//---------------------------------------------------------------------------------------------------------------
//
//  HAUD 2024.04.16
//
//
//
//---------------------------------------------------------------------------------------------------------------
// This SOFTWARE is provided as an Exemple by THE PROVIDER "as is" and "with all faults." THE PROVIDER makes no 
// representations or warranties of any kind concerning the safety, suitability, lack of viruses, inaccuracies, 
// typographical errors, or other harmful components of this SOFTWARE. There are inherent dangers in the use of 
// any software, and you are solely responsible for determining whether this SOFTWARE is compatible with your 
// equipment and other software installed on your equipment. You are also solely responsible for the protection 
// of your equipment and backup of your data, and THE PROVIDER will not be liable for any damages you may suffer 
// in connection with using, modifying, or distributing this SOFTWARE.
//---------------------------------------------------------------------------------------------------------------
FUNCTION_BLOCK fb_Mover
VAR
  _nMoverId         : UINT;

  _sState           : STRING;

  _Mover            : REFERENCE TO Tc3_Mc3PlanarMotion.MC_PlanarMover;
  _Feedback         : REFERENCE TO Tc3_Mc3PlanarMotion.MC_PlanarFeedback;

  // mover compact axis information
  _stInfo           : REFERENCE TO ST_MOVER_INFO; // ActPos, Enable, ...

  _bError           : BOOL;   // used in Cycle()
  _nErrorIdMover,             // used in Cycle()
  _nErrorIdPower    : UDINT;  // used in Cycle()

  //---------------------------------------------------------------------------
  // 
  //---------------------------------------------------------------------------
  _wMoverState      : DWORD;

END_VAR

METHOD Check : BOOL
// check The thing that should not be

IF NOT (_nMoverId > 0)
THEN
  _sState                     := 'Mover: missing ID';
  RETURN;
END_IF

IF NOT __ISVALIDREF(_Mover)
THEN
  _sState                     := 'Mover: missing pointer';
  RETURN;
END_IF

IF NOT __ISVALIDREF(_stInfo)
THEN
  _sState                     := '_stInfo: missing pointer';
  RETURN;
END_IF

_sState                       := 'CHECK_DONE';
Check                         := TRUE;
END_METHOD

METHOD Cycle : E_PROGRESS
VAR_INST
  _eState             : E_PROGRESS;

  _rtrigMoverError,
  _rtrigPowerError    : Tc2_Standard.R_TRIG;
END_VAR
IF NOT Check() THEN Cycle := E_PROGRESS.PROGRESS_ERROR; RETURN; END_IF

//-----------------------------------------------------------------------------------------------
// cyclic NC mapping
//-----------------------------------------------------------------------------------------------
_Mover.Update();
_Feedback.Update();
//-----------------------------------------------------------------------------------------------


//-----------------------------------------------------------------------------------------------
// cyclic error
//-----------------------------------------------------------------------------------------------

_rtrigPowerError(CLK := _Feedback.Error);

IF _rtrigMoverError.Q
THEN
  _bError                 := TRUE;  // deleted by Reset()
  // catch error
  _nErrorIdMover          := _Feedback.ErrorId;
  _stInfo.nErrorId        := _nErrorIdMover;
END_IF
//-----------------------------------------------------------------------------------------------

//-----------------------------------------------------------------------------------------------
// cyclic state
//-----------------------------------------------------------------------------------------------
IF NOT (_Mover.MCTOPLC.STD.State = MC_PLANAR_STATE.Enabled)
THEN
  _eState                       := E_PROGRESS.PROGRESS_INIT;
ELSE
  _eState                       := E_PROGRESS.PROGRESS_WORKING;
END_IF
 
IF _bError
THEN
  _eState                       := E_PROGRESS.PROGRESS_ERROR;
END_IF
//-----------------------------------------------------------------------------------------------


//-----------------------------------------------------------------------------
// cyclic Mover info data
// get collision avoiding information from cyclic interface
//-----------------------------------------------------------------------------------------------
_stInfo.bMoverEnabled           := (_Mover.MCTOPLC.STD.State = MC_PLANAR_STATE.Enabled);
_stInfo.bMoverStandstill        := NOT (_Mover.MCTOPLC.STD.Busy.BusyXYC);
_stInfo.bMoverError             := _bError;

_stInfo.rActPos.x               := _Mover.MCTOPLC.ACT.ActPos.x;
_stInfo.rActPos.y               := _Mover.MCTOPLC.ACT.ActPos.y;
_stInfo.rActPos.c               := _Mover.MCTOPLC.ACT.ActPos.c;
                                
_stInfo.rActPosX                := _Mover.MCTOPLC.ACT.ActPos.x;
_stInfo.rActPosY                := _Mover.MCTOPLC.ACT.ActPos.y;
_stInfo.rActPosC                := _Mover.MCTOPLC.ACT.ActPos.c;
                                
_stInfo.rActPosZ                := _Mover.MCTOPLC.ACT.ActPos.z;
                                
_stInfo.rActVeloX               := _Mover.MCTOPLC.ACT.ActVelo.x;
_stInfo.rActVeloY               := _Mover.MCTOPLC.ACT.ActVelo.y;
_stInfo.rActVeloZ               := _Mover.MCTOPLC.ACT.ActVelo.z;
_stInfo.rActVeloC               := _Mover.MCTOPLC.ACT.ActVelo.c;
//-----------------------------------------------------------------------------

Cycle                           := _eState;
END_METHOD

METHOD Disable : E_PROGRESS
VAR_INPUT
  Execute             : BOOL;
END_VAR
VAR_INST
  _nErrorId           : UDINT;
  _eState             : E_PROGRESS;
END_VAR
IF NOT Execute THEN _eState  := E_PROGRESS.PROGRESS_INIT; END_IF 
IF NOT Check() THEN Disable  := E_PROGRESS.PROGRESS_ERROR; RETURN; END_IF


CASE _eState
OF
  E_PROGRESS.PROGRESS_INIT:
    IF Execute
    THEN
      _nErrorId               := 0;
      _eState                 := E_PROGRESS.PROGRESS_BUSY;
    END_IF
END_CASE
//-----------------------------------------------------------------------------
//-----------------------------------------------------------------------------
CASE _eState
OF
  E_PROGRESS.PROGRESS_BUSY:
    _eState                   := E_PROGRESS.PROGRESS_PREPARE;
    _Mover.Disable(_Feedback);
END_CASE
//-----------------------------------------------------------------------------
//-----------------------------------------------------------------------------
CASE _eState
OF
  E_PROGRESS.PROGRESS_PREPARE:
    IF (_Mover.MCTOPLC.STD.State = MC_PLANAR_STATE.Disabled)
    THEN
      IF _Feedback.Error
      THEN
        _eState                 := E_PROGRESS.PROGRESS_ERROR;
      ELSIF _Feedback.Done
      THEN
        _eState                 := E_PROGRESS.PROGRESS_DONE;
      END_IF
    END_IF
END_CASE
//-----------------------------------------------------------------------------
//-----------------------------------------------------------------------------

Disable                       := _eState;
END_METHOD

METHOD Enable : E_PROGRESS
VAR_INPUT
  Execute             : BOOL;
END_VAR
VAR_INST
  _nErrorId           : UDINT;
  _eState             : E_PROGRESS;
END_VAR
IF NOT Execute THEN _eState  := E_PROGRESS.PROGRESS_INIT; END_IF 
IF NOT Check() THEN Enable   := E_PROGRESS.PROGRESS_ERROR; RETURN; END_IF


CASE _eState
OF
  E_PROGRESS.PROGRESS_INIT:
    IF Execute
    THEN
      _nErrorId               := 0;
      _eState                 := E_PROGRESS.PROGRESS_BUSY;
    END_IF
END_CASE
//-----------------------------------------------------------------------------
//-----------------------------------------------------------------------------
CASE _eState
OF
  E_PROGRESS.PROGRESS_BUSY:
    _eState                   := E_PROGRESS.PROGRESS_PREPARE;
    _Mover.Enable(_Feedback);
END_CASE
//-----------------------------------------------------------------------------
//-----------------------------------------------------------------------------
CASE _eState
OF
  E_PROGRESS.PROGRESS_PREPARE:
    IF (_Mover.MCTOPLC.STD.State = MC_PLANAR_STATE.Enabled)
    THEN
      IF _Feedback.Error
      THEN
        _eState                 := E_PROGRESS.PROGRESS_ERROR;
      ELSIF _Feedback.Done
      THEN
        _eState                 := E_PROGRESS.PROGRESS_DONE;
      END_IF
    ELSIF (_Mover.MCTOPLC.STD.State = MC_PLANAR_STATE.Error)
    THEN
      _eState                   := E_PROGRESS.PROGRESS_ERROR;
    END_IF
END_CASE
//-----------------------------------------------------------------------------
//-----------------------------------------------------------------------------

Enable                   := _eState;
END_METHOD

PROPERTY Feedback : reference to Tc3_Mc3PlanarMotion.MC_PlanarFeedback
SET
_Feedback REF= Feedback;
END_SET
END_PROPERTY

METHOD Halt : E_PROGRESS
VAR_INPUT
  Execute             : BOOL;
  stMoveData          : ST_MOVE_DATA;
END_VAR
VAR_INST
  _nErrorId           : UDINT;
  _eState             : E_PROGRESS;

	_Position           : Tc3_Physics.PositionXYC;
	_Constraint         : Tc3_Physics.DynamicConstraint_PathXY;
	_Options            : Tc3_Mc3PlanarMotion.ST_MoveToPositionOptions;
	_OptionsC           : ST_MoveCOptions;
END_VAR
IF NOT Execute 
THEN 
	_eState := E_PROGRESS.PROGRESS_INIT; 
END_IF 
IF NOT Check() 
THEN 
	Halt := E_PROGRESS.PROGRESS_ERROR; 
	RETURN; 
END_IF


CASE _eState
OF
  E_PROGRESS.PROGRESS_INIT:
    IF Execute
    THEN
      _nErrorId               := 0;
      _eState                 := E_PROGRESS.PROGRESS_BUSY;
    END_IF
END_CASE
//-----------------------------------------------------------------------------
//-----------------------------------------------------------------------------
CASE _eState
OF
  E_PROGRESS.PROGRESS_BUSY:
    _eState                     := E_PROGRESS.PROGRESS_PREPARE;
		_Position.SetValuesXYC(
                            x   := stMoveData.rPos.x,
													  y   := stMoveData.rPos.y,
                            c	  := 0.0);
								
		_Constraint.SetValuesVADJ(
                            V   := stMoveData.rVelo, 
                            A   := stMoveData.rAcc, 
                            D   := stMoveData.rAcc, 
                            J   := stMoveData.rJerk);

		_Options.useOrientation	    := FALSE;
END_CASE
//-----------------------------------------------------------------------------
//-----------------------------------------------------------------------------
CASE _eState
OF
  E_PROGRESS.PROGRESS_PREPARE:
    _eState                     := E_PROGRESS.PROGRESS_STARTUP;
    _Mover.Halt(_Feedback, _Constraint); 
END_CASE
//-----------------------------------------------------------------------------
//-----------------------------------------------------------------------------
CASE _eState
OF
  E_PROGRESS.PROGRESS_STARTUP:
    IF _Feedback.Error
    THEN
      _nErrorId                 := _feedback.ErrorId;
      _stInfo.nErrorId          := _nErrorId;

      _eState                   := E_PROGRESS.PROGRESS_ERROR;
    ELSIF _Feedback.Done
    THEN
      _eState                   := E_PROGRESS.PROGRESS_DONE;
    END_IF
END_CASE
//-----------------------------------------------------------------------------
//-----------------------------------------------------------------------------

Halt                          := _eState;
END_METHOD

PROPERTY Mover : REFERENCE to Tc3_Mc3PlanarMotion.MC_PlanarMover
SET
_Mover REF= Mover;
END_SET
END_PROPERTY

PROPERTY MoverId : uint
SET
_nMoverId := MoverId;
END_SET
END_PROPERTY

PROPERTY MoverInfo : REFERENCE to ST_MOVER_INFO
SET


	_stInfo ref= MoverInfo;
END_SET
END_PROPERTY

METHOD MoveToPos : E_PROGRESS
VAR_INPUT
  Execute             : BOOL;
  stMoveData          : ST_MOVE_DATA;
END_VAR
VAR_INST
  _nErrorId           : UDINT;
  _rDelta,
  _rPos               : LREAL;
  _eState             : E_PROGRESS;

	_Position           : Tc3_Physics.PositionXYC;
	_Constraint         : Tc3_Physics.DynamicConstraint_PathXY;
  _ConstraintC        : Tc3_Physics.DynamicConstraint_PathXY;
	_Options            : Tc3_Mc3PlanarMotion.ST_MoveToPositionOptions;
	_OptionsC           : ST_MoveCOptions;

  _rTmpV,
  _rTmpA,
  _rTmpD,
  _rTmpJ              : LREAL;
END_VAR
IF NOT Execute THEN _eState  := E_PROGRESS.PROGRESS_INIT; END_IF 
IF NOT Check() THEN MoveToPos   := E_PROGRESS.PROGRESS_ERROR; RETURN; END_IF


CASE _eState
OF
  E_PROGRESS.PROGRESS_INIT:
    IF Execute
    THEN
      _nErrorId                 := 0;
      _rDelta                   := SEL((stMoveData.rDelta < 0.01), stMoveData.rDelta, 0.05);
      _eState                   := E_PROGRESS.PROGRESS_BUSY;

      _rTmpV   := stMoveData.rVelo/10.0; 
      _rTmpA   := stMoveData.rAcc/10.0;
      _rTmpD   := stMoveData.rAcc/10.0; 
      _rTmpJ   := stMoveData.rJerk/10.0;


		  _Constraint.SetValuesVADJ(
                            V   := _rTmpV, 
                            A   := _rTmpA, 
                            D   := _rTmpD, 
                            J   := _rTmpJ);
  
      _Mover.MoveZ(
            commandFeedback     := _Feedback, 
            targetPosition      := stMoveData.rPosZ,
            constraint          := _Constraint);

		  _Options.useOrientation	  := FALSE;
    END_IF
END_CASE
//-----------------------------------------------------------------------------
//-----------------------------------------------------------------------------
CASE _eState
OF
  E_PROGRESS.PROGRESS_BUSY:
    IF _Feedback.Error OR _Feedback.Aborted
    THEN
      _nErrorId                 := _feedback.ErrorId;
      _stInfo.nErrorId          := _nErrorId;

      _eState                   := E_PROGRESS.PROGRESS_ERROR;

    ELSIF _Feedback.Done OR NOT _Feedback.Busy
    THEN
      _eState                   := E_PROGRESS.PROGRESS_PREPARE;

      IF (stMoveData.nAxisFirst = 1)
      THEN
        _Position.SetValuesXYC(
                            x   := stMoveData.rPos.x,
                            y   := _Mover.MCTOPLC.SET.SetPos.y,
                            c	  := 0.0);

      ELSIF (stMoveData.nAxisFirst = 2)
      THEN
        _Position.SetValuesXYC(
                            x   := _Mover.MCTOPLC.SET.SetPos.x,
                            y   := stMoveData.rPos.y,
                            c	  := 0.0);
      ELSE
        _Position.SetValuesXYC(
                            x   := stMoveData.rPos.x,
                            y   := stMoveData.rPos.y,
                            c	  := 0.0);
      END_IF								

		  _Options.useOrientation	  := FALSE;
    END_IF

  E_PROGRESS.PROGRESS_PREPARE:
    _eState                     := E_PROGRESS.PROGRESS_STARTUP;
		  _Options.useOrientation	  := FALSE;

		  _Constraint.SetValuesVADJ(
                            V   := stMoveData.rVelo, 
                            A   := stMoveData.rAcc, 
                            D   := stMoveData.rAcc, 
                            J   := stMoveData.rJerk);


		_Mover.MoveToPosition(
            commandFeedback     := _Feedback, 
            targetPosition      := _Position, 
            constraint          := _Constraint, 
            options             := _Options);

END_CASE
//-----------------------------------------------------------------------------
//-----------------------------------------------------------------------------
CASE _eState
OF
  E_PROGRESS.PROGRESS_STARTUP:
    IF _Feedback.Error OR _Feedback.Aborted
    THEN
      _nErrorId                 := _Feedback.ErrorId;
      _stInfo.nErrorId          := _nErrorId;

      _eState                   := E_PROGRESS.PROGRESS_ERROR;

    ELSIF _Feedback.Done  OR NOT _Feedback.Busy
    THEN

      IF (stMoveData.nAxisFirst = 1)
      THEN
        _eState                 := E_PROGRESS.PROGRESS_CHECK;
        _Position.SetValuesXYC(
                            x   := _Mover.MCTOPLC.ACT.ActPos.x,
                            y   := stMoveData.rPos.y,
                            c	  := 0.0);

      ELSIF (stMoveData.nAxisFirst = 2)
      THEN
        _eState                 := E_PROGRESS.PROGRESS_CHECK;
        _Position.SetValuesXYC(
                            x   := stMoveData.rPos.x,
                            y   := _Mover.MCTOPLC.ACT.ActPos.y,
                            c	  := 0.0);
      ELSE
        _eState                 := E_PROGRESS.PROGRESS_WORKING;

      END_IF								

		  _Options.useOrientation	  := FALSE;
    END_IF

  E_PROGRESS.PROGRESS_CHECK:
    _eState                     := E_PROGRESS.PROGRESS_OCCUPIED;
		  _Options.useOrientation	  := FALSE;

		  _Constraint.SetValuesVADJ(
                            V   := stMoveData.rVelo, 
                            A   := stMoveData.rAcc, 
                            D   := stMoveData.rAcc, 
                            J   := stMoveData.rJerk);


		_Mover.MoveToPosition(
            commandFeedback     := _Feedback, 
            targetPosition      := _Position, 
            constraint          := _Constraint, 
            options             := _Options);

END_CASE
//-----------------------------------------------------------------------------
//-----------------------------------------------------------------------------
CASE _eState
OF
  E_PROGRESS.PROGRESS_OCCUPIED:
    IF _Feedback.Error OR _Feedback.Aborted
    THEN
      _nErrorId                 := _Feedback.ErrorId;
      _stInfo.nErrorId          := _nErrorId;

      _eState                   := E_PROGRESS.PROGRESS_ERROR;

    ELSIF _Feedback.Done OR NOT _Feedback.Busy
    THEN
      _eState                   := E_PROGRESS.PROGRESS_WORKING;
		  _Options.useOrientation	  := FALSE;
    END_IF
END_CASE
//-----------------------------------------------------------------------------
//-----------------------------------------------------------------------------
CASE _eState
OF
  E_PROGRESS.PROGRESS_WORKING:
    _eState                     := E_PROGRESS.PROGRESS_STILL_WORKING;

        _rTmpV   := stMoveData.rVelo/10.0; 
        _rTmpA   := stMoveData.rAcc/10.0;
        _rTmpD   := stMoveData.rAcc/10.0; 
        _rTmpJ   := stMoveData.rJerk/10.0;
  
        _ConstraintC.SetValuesVADJ(
                            V   := _rTmpV, 
                            A   := _rTmpA, 
                            D   := _rTmpD, 
                            J   := _rTmpJ);

    _OptionsC.additionalTurns   := 0;
    _OptionsC.direction         := stMoveData.rPos.cDirection;;

    _Mover.MoveC(
            commandFeedback     := _Feedback, 
            targetPosition      := stMoveData.rPos.c,
            constraint          := _ConstraintC,
            options             := _OptionsC);
END_CASE
//-----------------------------------------------------------------------------
//-----------------------------------------------------------------------------
CASE _eState
OF
  E_PROGRESS.PROGRESS_STILL_WORKING:
    IF _Feedback.Error OR _Feedback.Aborted
    THEN
      _nErrorId                 := _Feedback.ErrorId;
      _stInfo.nErrorId          := _nErrorId;

      _eState                   := E_PROGRESS.PROGRESS_ERROR;

    ELSIF _Feedback.Done OR NOT _Feedback.Busy
    THEN
      IF (_stInfo.rActPosC < stMoveData.rPos.c + 0.02) AND
         (_stInfo.rActPosC > stMoveData.rPos.c - 0.02)
      THEN
        _eState                  := E_PROGRESS.PROGRESS_DONE;
      END_IF
    END_IF
END_CASE
//-----------------------------------------------------------------------------
//-----------------------------------------------------------------------------
MoveToPos                       := _eState;
//-----------------------------------------------------------------------------
//-----------------------------------------------------------------------------
END_METHOD

METHOD Reset : E_PROGRESS
VAR_INPUT
  Execute             : BOOL;
END_VAR
VAR_INST
  _nErrorId           : UDINT;
  _eState             : E_PROGRESS;
END_VAR
IF NOT Execute THEN _eState  := E_PROGRESS.PROGRESS_INIT; END_IF 
IF NOT Check() THEN Reset    := E_PROGRESS.PROGRESS_ERROR; RETURN; END_IF


CASE _eState
OF
  E_PROGRESS.PROGRESS_INIT:
    IF Execute
    THEN
      _stInfo.nErrorId        :=
      _nErrorId               := 0;
      _eState                 := E_PROGRESS.PROGRESS_BUSY;
    END_IF
END_CASE
//-----------------------------------------------------------------------------
//-----------------------------------------------------------------------------
CASE _eState
OF
  E_PROGRESS.PROGRESS_BUSY:
    _eState                   := E_PROGRESS.PROGRESS_PREPARE;
    _Mover.Reset(_Feedback);
END_CASE
//-----------------------------------------------------------------------------
//-----------------------------------------------------------------------------
CASE _eState
OF
  E_PROGRESS.PROGRESS_PREPARE:
    IF _Feedback.Error
    THEN
      _nErrorId               := _Feedback.ErrorId;
      _stInfo.nErrorId        := _nErrorId;

      _eState                 := E_PROGRESS.PROGRESS_ERROR;

    ELSIF _Feedback.Done
    THEN
      _eState                 := E_PROGRESS.PROGRESS_DONE;
    END_IF
END_CASE
//-----------------------------------------------------------------------------
//-----------------------------------------------------------------------------

Reset                         := _eState;
END_METHOD

END_FUNCTION_BLOCK

(* stored: Version 1.1.0.1, ProductVersion 3.1.4024.13
   POU fb_Mover: Id {0329c584-f72c-48ef-81e9-d36f2b915502}, SpecialFunc None
   Folder methods: Id {d4f48e59-bafb-4a6b-a547-9f57a3dde1b3}
   Folder properties: Id {9b756c45-f31b-4fd8-944d-37c13ea518e9}
   Method Check: Id {7aad3024-4d91-4070-bd1c-7ab21c07b418}
   Method Cycle: Id {23c9e7eb-0f59-4742-a92e-59fc57018459}
   Method Disable: Id {097d7d29-677b-4897-9517-c610ca359790}
   Method Enable: Id {5c42fddf-2f46-4658-9cfe-4e104b612772}
   Property Feedback: Id {0b7b91b5-ce48-4dd5-9886-b74e22e39ef2}
   Set Set: Id {1e5b18f4-7ef6-4a39-b3b1-129db4f4e8b6}
   Method Halt: Id {6d1913d1-ebf7-491a-a13e-d4ef262d26ef}
   Property Mover: Id {725f2a78-1f2c-4af9-8ce5-bb55abd5bdc7}
   Set Set: Id {f63f36af-a1b3-44d0-911f-8078223fe58a}
   Property MoverId: Id {0ba03e0e-28d1-4142-b9f5-7e4ec07c6988}
   Set Set: Id {c36f4173-a354-4b08-9d63-481abb7f409a}
   Property MoverInfo: Id {37db38a4-3c3d-40a1-a24e-7c3e5a8f6c0d}
   Set Set: Id {09a628eb-fb2a-4de3-b247-fb2dd797a92f}
   Method MoveToPos: Id {fb779f0f-ad18-4dac-8c8b-6a09fac8cfc2}
   Method Reset: Id {f267dfd0-7a70-4720-839c-88e90bbf285e} *)
